(* Logix 5000 project; controller RSL5k_18_Template_noLib Emulate 5570 rev 32.11; software revision 32.02; part 9 of 16 *)
(* tags used below, declared in another part *)
   Inp_CascSP : ALIAS FOR Wrk_PIDE.SPCascade;   // Setpoint in Cascade, Independent PV in Ratio (PVEU)
   Inp_FF : REAL;   // FeedForward term (CVEU)
   Inp_FFPrev : REAL;   // Previous scan FF term (CVEU)
   Inp_CVInitVal : ALIAS FOR Wrk_PIDE.CVInitValue;   // Value to Initialize the CV to when requested (CVRaw)
   Inp_CVPrev : REAL;   // Previous scan CV (CVEU)
   Inp_UseCVInitVal : ALIAS FOR Wrk_PIDE.CVInitReq;   // 1=Initialize CV to Inp_CVInitValue
   Inp_HandFdbk : REAL;   // CV Feedback used in Hand Mode (CVEU)
   Inp_OvrdRatio : REAL;   // Loop Ratio in Override (unitless)
   Inp_OvrdSP : REAL;   // Loop Auto Setpoint (SP) in Override (PVEU)
   Inp_OvrdCV : REAL;   // Loop Manual Output (CV) in Override (CVEU)
   Inp_OvrdSPRoCLimInc : REAL;   // Override Setting for Setpoint Positive Rate of Change Limit (PVEU/sec)
   Inp_OvrdSPRoCLimDec : REAL;   // Override Setting for Setpoint Negative Rate of Change Limit (PVEU/sec)
   Cfg_HasRatio : ALIAS FOR Wrk_PIDE.UseRatio;   // 1=Casc Loop Mode is Ratio, 0=Casc Loop Mode is Cascade
   Cfg_PVTrack : ALIAS FOR Wrk_PIDE.PVTracking;   // 1=SP tracks PV in Manual, 0=no PV tracking
   Cfg_LimitManCV : ALIAS FOR Wrk_PIDE.CVManLimiting;   // 1=CV limits enforced in Manual, 0=No CV Limiting in Manual
   Cfg_SetTrack : BOOL;   // 1=Prog/Oper/Ext Settings track, 0=no Settings tracking
   Cfg_SetTrackOvrdHand : BOOL;   // 1=Prog/Oper/Ext Settings track Override/Hand Inputs (CV, SP, Ratio)
   Cfg_SkipSPRoCLim : BOOL;   // 1=Skip SP RoC Limiting in Intlk, Maint, Ovrd
   Cfg_NormLM : DINT;   // Normal Loop Mode 0=Disable Normal selection, 1=Man, 2=Auto, 3=Casc
   Cfg_PwrupLM : DINT;   // Powerup Loop Mode 0=No change (last), 1=Man (w/ CV), 2=Auto (w/ SP), 3=Casc, 4=Normal
   Cfg_IntlkTripCVAct : DINT;   // Interlock Trip CV Action: 0=none, 1=hold last good, 2=use Cfg_IntlkCV
   Cfg_SPFailCVAct : DINT;   // SP Fail CV Action: 0=none, 1=hold last good, 2=use Cfg_IntlkCV
   Cfg_PVFailCVAct : DINT;   // PV Fail CV Action: 1=hold last good, 2=use Cfg_IntlkCV
   Cfg_CVFailCVAct : DINT;   // CV Fail CV Action: 1=hold last good, 2=use Cfg_IntlkCV
   Cfg_MinSP : ALIAS FOR Wrk_PIDE.SPLLimit;   // Minimum allowed Setpoint (SP) (PVEU)
   Cfg_MaxSP : ALIAS FOR Wrk_PIDE.SPHLimit;   // Maximum allowed Setpoint (SP) (PVEU)
   Cfg_MaxSPRoCInc : REAL;   // Maximum allowed Setpoint Positive Rate of Change Limit (PVEU/sec)
   Cfg_MaxSPRoCDec : REAL;   // Maximum allowed Setpoint Negative Rate of Change Limit (PVEU/sec)
   Cfg_SPRampMaxDev : REAL;   // If deviation exceeds this value, pause SP ramp (0.0=never pause) (PVEU)
   Cfg_PVEUMin : ALIAS FOR Wrk_PIDE.PVEUMin;   // PV Engineering Units Mimimum Value (PVEU)
   Cfg_PVEUMax : ALIAS FOR Wrk_PIDE.PVEUMax;   // PV Engineering Units Maximum Value (PVEU)
   Cfg_CVEUMin : REAL;   // CV Engineering Units Minimum Value (CVEU)
   Cfg_CVEUMax : REAL;   // CV Engineering Units Maximum Value (CVEU)
   Cfg_CVRawMin : ALIAS FOR Wrk_PIDE.CVEUMin;   // CV Output Units Minimum Value (CVRaw, for scaling))
   Cfg_CVRawMax : ALIAS FOR Wrk_PIDE.CVEUMax;   // CV Output Units Maximum Value (CVRaw, for scaling)
   Cfg_ExecT : REAL;   // Execution Time (interval) for PID Algorithm (sec)
   Cfg_MinCV : REAL;   // Minimum allowed Controlled Variable (CV) value (CVEU)
   Cfg_MaxCV : REAL;   // Maximum allowed Controlled Variable (CV) value (CVEU)
   Cfg_CVRoCLim : REAL;   // CV Rate of Change Limit (CVEU/sec)
   Cfg_MaxInactiveCV : REAL;   // When Val_CV is greater than this value, set Sts_Active (for HMI) (CVEU)
   Cfg_IntlkCV : REAL;   // CV Value to use with Interlock / Bad Value CV action (CVEU)
   Cfg_PwrupCV : REAL;   // Loop CV on powerup, used if Cfg_PwrupLM <> 0 (none) (CVEU)
   PSet_Ratio : REAL;   // Program Setting for Ratio (loop CasRat and Ratio enabled) (unitless)
   PSet_SP : REAL;   // Program Setting for Setpoint (loop Auto) (PVEU)
   PSet_SPRoCLimInc : REAL;   // Program Setting for Setpoint Rate of Change Limit Increasing (PVEU/sec)
   PSet_SPRoCLimDec : REAL;   // Program Setting for Setpoint Rate of Change Limit Decreasing (PVEU/sec)
   PSet_CV : REAL;   // Program Setting for Controlled Variable (loop Manual) (CVEU)
   XSet_Ratio : REAL;   // External Setting for Ratio (loop CasRat and Ratio enabled) (unitless)
   XSet_SP : REAL;   // External Setting for Setpoint (loop Auto) (PVEU)
   XSet_SPRoCLimInc : REAL;   // External Setting for Setpoint Rate of Change Limit Increasing (PVEU/sec)
   XSet_SPRoCLimDec : REAL;   // External Setting for Setpoint Rate of Change Limit Decreasing (PVEU/sec)
   XSet_CV : REAL;   // External Setting for Controlled Variable (loop Manual) (CVEU)
   Out_CV : ALIAS FOR Wrk_PIDE.CVEU;   // CV to final control element (CV Raw Units)
   Val_PV : REAL;   // Value of Loop PV (PVEU)
   Val_Ratio : ALIAS FOR Wrk_PIDE.Ratio;   // Value of Loop Ratio (unitless)
   Val_SPSet : REAL;   // Value of selected SP (before clamping and ramping) (PVEU)
   Val_SPRoCInc : REAL;   // Current Value of Setpoint Rate of Change Limit Increasing (PVEU/sec)
   Val_SPRoCDec : REAL;   // Current Value of Setpoint Rate of Change Limit Decreasing (PVEU/sec)
   Val_E : ALIAS FOR Wrk_PIDE.E;   // Loop Error (PV-SP) (PVEU)
   Val_CVSet : REAL;   // Value of selected CV (before clamping and ramping) (CVEU)
   Val_CVOut : REAL;   // Value of CV Output (after ramping and clamping (CVEU)
   Val_ActExecT : ALIAS FOR Wrk_PIDE.DeltaT;   // Actual PID Algorithm Execution Time (Interval) (sec)
   Val_Init : REAL;   // Initialization Value for this loop's Cascade Primary (PVEU)
   Val_PVEUMin : REAL;   // Minimum of PV scaled range (PVEU)
   Val_PVEUMax : REAL;   // Maximum of PV scaled range (PVEU)
   Val_CVEUMin : REAL;   // Minimum of CV scaled range (CVEU)
   Val_CVEUMax : REAL;   // Maximum of CV scaled range (CVEU)
   Sts_InstrFaults1 : DINT;   // PIDE Block Status1 Instruction Fault bits (See PIDE Instruction Help)
   Sts_InstrFaults2 : DINT;   // PIDE Block Status2 Instruction Fault bits (See PIDE Instruction Help)
   Sts_Casc : BOOL;   // 1=Loop Mode is Cascade/Ratio
   Sts_Auto : BOOL;   // 1=Loop Mode is Auto
   Sts_Man : BOOL;   // 1=Loop Mode is Manual
   Sts_NormLM : BOOL;   // 1=Loop is in Normal Loop Mode (see Cfg_NormLM)
   Sts_InitReq : BOOL;   // 1=CV Initialize Request to this loop's Primary
   Sts_RatioClamped : BOOL;   // 1=Selected Ratio (PSet/OSet_Ratio or Inp_OvrdRatio) has been clamped
   Sts_SPBad : ALIAS FOR Wrk_PIDE.SPProgInv;   // 1=SP Value is Bad (quality) or invalid or Casc SP comms fault
   Sts_IntlkSP : BOOL;   // 1=SP Value is being set by shed to Interlock SP
   Sts_SPHeld : BOOL;   // 1=SP Value is being set by shed to hold last good SP
   Sts_SPShed : BOOL;   // 1=SP from Shed, 0=SP from Prog, Oper, Ovrd (A), Casc SP Input (C) or PV Track (M)
   Sts_SPTrackPV : BOOL;   // 1=SP Value is being set by PV Tracking (in Manual Mode)
   Sts_SPClamped : BOOL;   // 1=Selected SP is being clamped (for faceplate animation)
   Sts_SPRamping : BOOL;   // 1=SP is ramping toward Val_SPSet, 0=ramp complete
   Sts_SkipSPRoCLim : BOOL;   // 1=SP rate limiting is being skipped (for faceplate animation)
   Sts_PVBad : BOOL;   // 1=PV Value, comms, quality or EU Limitis Bad
   Sts_CVBad : BOOL;   // 1=CV Value is Bad (quality) or invalid or CV comms fault
   Sts_IntlkCV : BOOL;   // 1=CV Value is being set by shed to Interlock CV
   Sts_CVHeld : BOOL;   // 1=CV Value is being set by shed to hold last good CV
   Sts_CVShed : BOOL;   // 1=CV from Shed, 0=CV from Prog, Oper, Ovrd (Man), or PID (Auto, Casc)
   Sts_CVClamped : BOOL;   // 1=Selected CV is being clamped (for faceplate animation)
   Sts_Active : BOOL;   // 1=CV is greater than Cfg_MaxInactiveCV, show graphic symbol as "active"
   Sts_Err : BOOL;   // 1=Error in Config: see detail Err bits for reason
   Err_Timer : BOOL;   // 1=Error in Config: Status On-Delay or Off-Delay Time Invalid
   Err_RatioLim : ALIAS FOR Wrk_PIDE.RatioLimitsInv;   // 1=Error in Config: Ratio Clamping Limits Invalid
   Err_SPLim : ALIAS FOR Wrk_PIDE.SPLimitsInv;   // 1=Error in Config: Setpoint Clamping Limits Invalid
   Err_CVLim : ALIAS FOR Wrk_PIDE.CVLimitsInv;   // 1=Error in Config: CV Clamping Limits Invalid
   Err_PVEU : ALIAS FOR Wrk_PIDE.PVSpanInv;   // 1=Error in Config: PV EU Max/Min Invalid
   Err_CVEU : BOOL;   // 1=Error in Config: CV EU Max/Min Invalid
   Sts_Hand : ALIAS FOR CmdSrc.Sts_Hand;
   Sts_OoS : ALIAS FOR CmdSrc.Sts_OoS;
   Sts_Maint : ALIAS FOR CmdSrc.Sts_Maint;
   Sts_Ovrd : ALIAS FOR CmdSrc.Sts_Ovrd;
   Sts_Fail : ALIAS FOR Fail.Inp;   // 1=Loop Failure: PV Bad, SP Bad or CV Comm Failure or Bad
   P_PIDE : BOOL;   // Unique Parameter Name for auto - discovery
   CmdSrc : P_CmdSrc;   // Control / Command Source Selection
   Fail : P_Alarm;   // Loop (SP, PV or CV) Failure Alarm
   Wrk_ScanTime : REAL;   // Time since previous scan (sec)
   Wrk_SPStepInc : REAL;   // Amount to add this scan for SP RoC increasing limiting (PVEU)
   Wrk_ScanT : TIMER;   // Scan Timer (milliseconds, always runs)
   Wrk_Casc : BOOL;   // Internal Loop Mode latch: Cascade selected
   Wrk_Auto : BOOL;   // Internal Loop Mode latch: 1=Auto selected
   Wrk_Man : BOOL;   // Internal Loop Mode latch: Manual selected
   Wrk_SPStepDec : REAL;   // Amount to add this scan for SP RoC decreasing limiting (PVEU)
   Wrk_IntlkTripShed : BOOL;   // Shed Latch for Interlock Not OK
   Wrk_PVFailShed : BOOL;   // Shed Latch for PV Failure
   Wrk_SPFailShed : BOOL;   // Shed Latch for SP Failure
   Wrk_CVFailShed : BOOL;   // Shed Latch for CV Failure
   Wrk_AlgoScanT : REAL;   // Time since last calculation of PID Algorithm (sec)
   Wrk_SkippedPID : BOOL;   // PID Algorithm was NOT scanned this time through
   LoLoDevGate : P_Gate;   // Low-Low Deviation Gate/Delay
   LoDevGate : P_Gate;   // Low Deviation Gate/Delay
   HiDevGate : P_Gate;   // High Deviation Gate/Delay
   HiHiDevGate : P_Gate;   // High-High Deviation Gate/Delay
   Wrk_PIDE : PID_ENHANCED;   // Built-in controller PID algorithm
   Wrk_Autotune : PIDE_AUTOTUNE;   // Autotune tag associated with built-in PID algorithm
   Wrk_PIDE_only : P_PIDE_only;   // Backing tag for AOI containing PIDE (with optional autotune)
   HMI_HasAutotune : BOOL;   // 1=P_PIDE_Only AOI has been modified to include Autotune par. on PIDE block
   OSet_CV : REAL;   // Operator Setting for Controlled Variable (loop Manual) (CVEU)
   OSet_SPRoCLimDec : REAL;   // Operator Setting for Setpoint Rate of Change Limit Decreasing (PVEU/sec)
   OSet_SPRoCLimInc : REAL;   // Operator Setting for Setpoint Rate of Change Limit Increasing (PVEU/sec)
   OSet_SP : REAL;   // Operator Setting for Setpoint (loop Auto) (PVEU)
   OSet_Ratio : REAL;   // Operator Setting for Ratio (loop CasRat and Ratio enabled) (unitless)
   Wrk_ExtHas : SINT;   // External owns: .0=LM, .1=CV, .2=SP, .3=Ratio
   Wrk_ProgHas : SINT;   // Program owns: .0=LM, .1=CV, .2=SP, .3=Ratio
   Wrk_OperHas : SINT;   // Operator owns: .0=LM, .1=CV, .2=SP, .3=Ratio
   ORdy_CV : BOOL;   // 1=Ready for OSet_CV (enables data entry field)
   ORdy_SP : BOOL;   // 1=Ready for OSet_SP (enables data entry field)
   Wrk_FirstPIDCalc : BOOL;   // PID Not Skipped ONS store
   ORdy_SPRoCLimInc : BOOL;   // 1=Ready for OSet_SPRoCLimInc (enables data entry field)
   ORdy_SPRoCLimDec : BOOL;   // 1=Ready for OSet_SPRoCLimDec (enables data entry field)
   Wrk_Init : BOOL;   // 1=AOI has been initialized
   Wrk_SPRoCLimDec : REAL;   // Actual SP Rate of Change Limit Decreasing
   Wrk_SPRoCLimInc : REAL;   // Actual SP Rate of Change Limit Increasing
   Wrk_SPRampBusy : BOOL;   // 1=SP Ramp Wizard ramp is in progress
   Wrk_RatioClamped : BOOL;   // Buffer for building Sts_RatioClamped
(* P_PIDE, continued *)

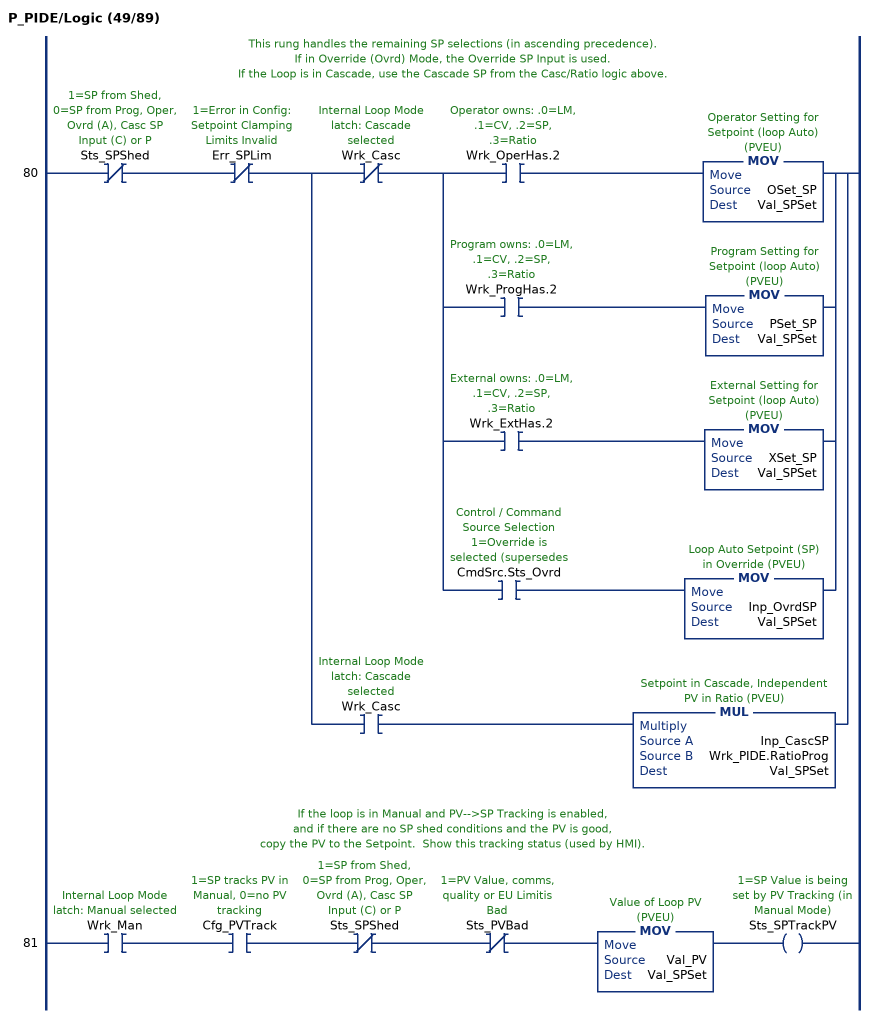
   [picture p175: P_PIDE/Logic rungs 80-81]
   // This rung handles the remaining SP selections (in ascending precedence).
   // If in Override (Ovrd) Mode, the Override SP Input is used.
   // If the Loop is in Cascade, use the Cascade SP from the Casc/Ratio logic above.
   80: XIO(Sts_SPShed)XIO(Err_SPLim)[XIO(Wrk_Casc) [XIC(Wrk_OperHas.2) MOV(OSet_SP,Val_SPSet) ,XIC(Wrk_ProgHas.2) MOV(PSet_SP,Val_SPSet) ,XIC(Wrk_ExtHas.2) MOV(XSet_SP,Val_SPSet) ,XIC(CmdSrc.Sts_Ovrd) MOV(Inp_OvrdSP,Val_SPSet) ] ,XIC(Wrk_Casc) MUL(Inp_CascSP,Wrk_PIDE.RatioProg,Val_SPSet) ];
   // If the loop is in Manual and PV-->SP Tracking is enabled,
   // and if there are no SP shed conditions and the PV is good,
   // copy the PV to the Setpoint.  Show this tracking status (used by HMI).
   81: XIC(Wrk_Man)XIC(Cfg_PVTrack)XIO(Sts_SPShed)XIO(Sts_PVBad)MOV(Val_PV,Val_SPSet)OTE(Sts_SPTrackPV);
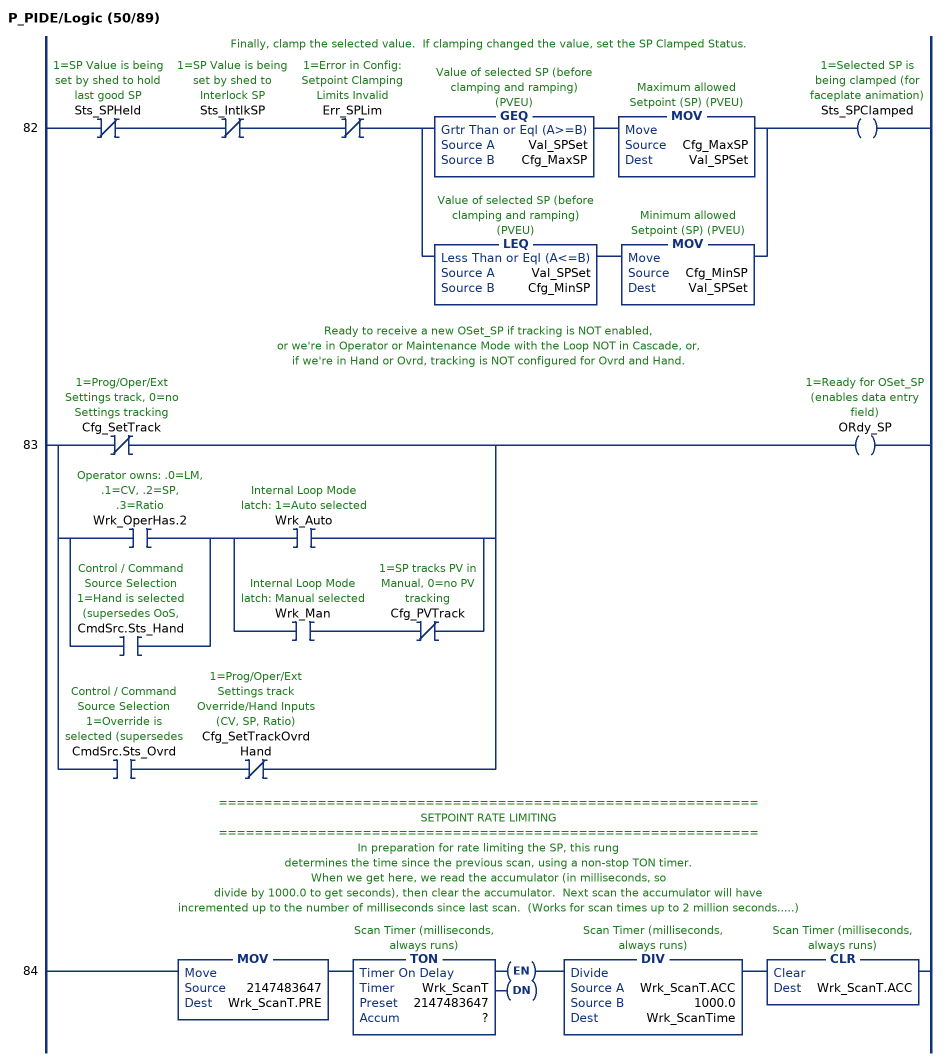
   // Finally, clamp the selected value.  If clamping changed the value, set the SP Clamped Status.
   82: XIO(Sts_SPHeld)XIO(Sts_IntlkSP)XIO(Err_SPLim)[GEQ(Val_SPSet,Cfg_MaxSP) MOV(Cfg_MaxSP,Val_SPSet) ,LEQ(Val_SPSet,Cfg_MinSP) MOV(Cfg_MinSP,Val_SPSet) ]OTE(Sts_SPClamped);
   // Ready to receive a new OSet_SP if tracking is NOT enabled,
   // or we're in Operator or Maintenance Mode with the Loop NOT in Cascade, or,
   // if we're in Hand or Ovrd, tracking is NOT configured for Ovrd and Hand.
   83: [XIO(Cfg_SetTrack) ,[XIC(Wrk_OperHas.2) ,XIC(CmdSrc.Sts_Hand) ] [XIC(Wrk_Auto) ,XIC(Wrk_Man) XIO(Cfg_PVTrack) ] ,XIC(CmdSrc.Sts_Ovrd) XIO(Cfg_SetTrackOvrdHand) ]OTE(ORdy_SP);
   // ============================================================
   // SETPOINT RATE LIMITING
   // ============================================================
   // In preparation for rate limiting the SP, this rung
   // determines the time since the previous scan, using a non-stop TON timer.
   // When we get here, we read the accumulator (in milliseconds, so
   // divide by 1000.0 to get seconds), then clear the accumulator.  Next scan the accumulator will have
   // incremented up to the number of milliseconds since last scan.  (Works for scan times up to 2 million seconds.....)
   84: MOV(2147483647,Wrk_ScanT.PRE)TON(Wrk_ScanT,?,?)DIV(Wrk_ScanT.ACC,1000.0,Wrk_ScanTime)CLR(Wrk_ScanT.ACC);
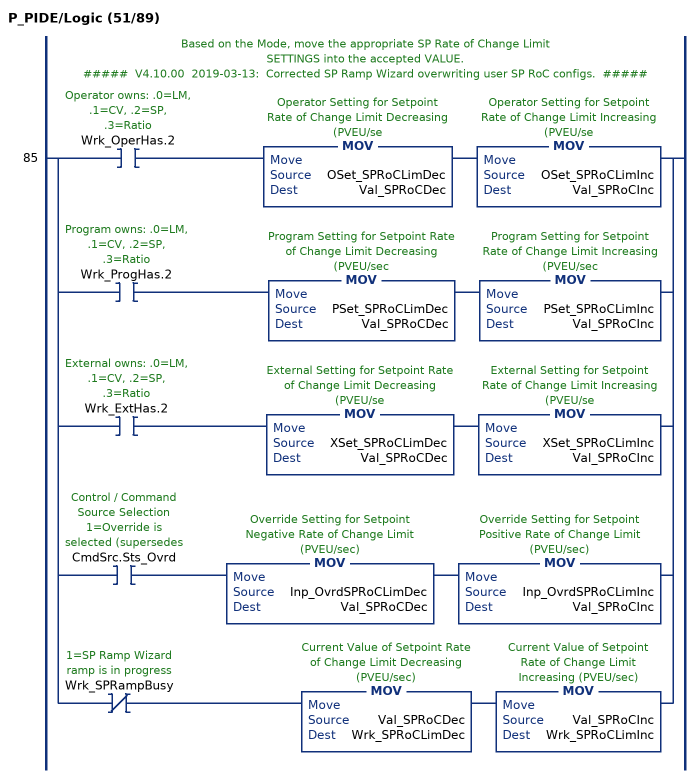
   // Based on the Mode, move the appropriate SP Rate of Change Limit
   // SETTINGS into the accepted VALUE.
   // #####  V4.10.00  2019-03-13:  Corrected SP Ramp Wizard overwriting user SP RoC configs.  #####
   85: [XIC(Wrk_OperHas.2) MOV(OSet_SPRoCLimDec,Val_SPRoCDec) MOV(OSet_SPRoCLimInc,Val_SPRoCInc) ,XIC(Wrk_ProgHas.2) MOV(PSet_SPRoCLimDec,Val_SPRoCDec) MOV(PSet_SPRoCLimInc,Val_SPRoCInc) ,XIC(Wrk_ExtHas.2) MOV(XSet_SPRoCLimDec,Val_SPRoCDec) MOV(XSet_SPRoCLimInc,Val_SPRoCInc) ,XIC(CmdSrc.Sts_Ovrd) MOV(Inp_OvrdSPRoCLimDec,Val_SPRoCDec) MOV(Inp_OvrdSPRoCLimInc,Val_SPRoCInc) ,XIO(Wrk_SPRampBusy) MOV(Val_SPRoCDec,Wrk_SPRoCLimDec) MOV(Val_SPRoCInc,Wrk_SPRoCLimInc) ];
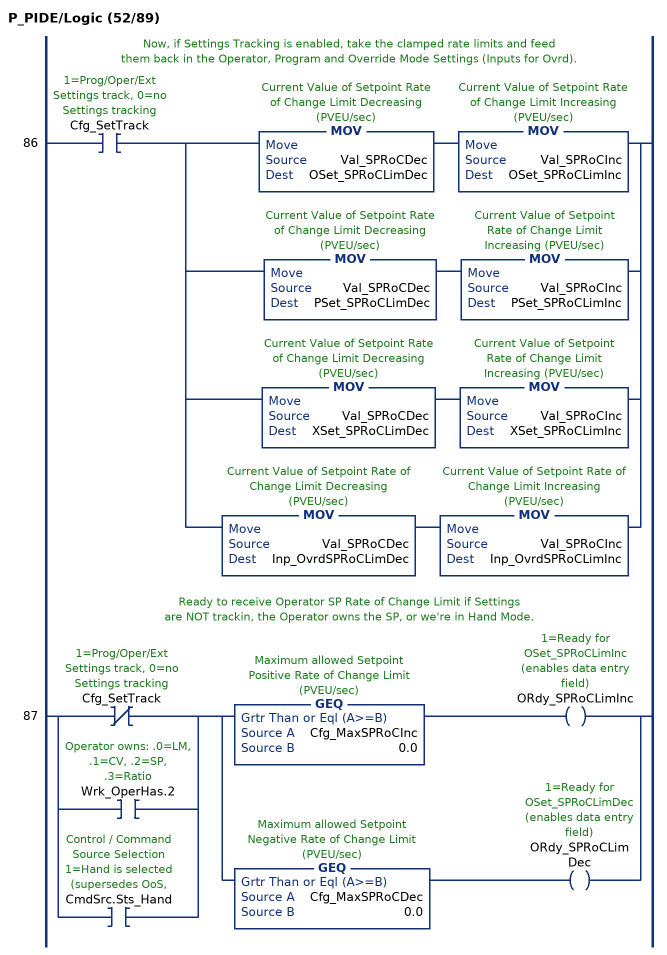
   // Now, if Settings Tracking is enabled, take the clamped rate limits and feed
   // them back in the Operator, Program and Override Mode Settings (Inputs for Ovrd).
   86: XIC(Cfg_SetTrack)[MOV(Val_SPRoCDec,OSet_SPRoCLimDec) MOV(Val_SPRoCInc,OSet_SPRoCLimInc) ,MOV(Val_SPRoCDec,PSet_SPRoCLimDec) MOV(Val_SPRoCInc,PSet_SPRoCLimInc) ,MOV(Val_SPRoCDec,XSet_SPRoCLimDec) MOV(Val_SPRoCInc,XSet_SPRoCLimInc) ,MOV(Val_SPRoCDec,Inp_OvrdSPRoCLimDec) MOV(Val_SPRoCInc,Inp_OvrdSPRoCLimInc) ];
   // Ready to receive Operator SP Rate of Change Limit if Settings
   // are NOT trackin, the Operator owns the SP, or we're in Hand Mode.
   87: [XIO(Cfg_SetTrack) ,XIC(Wrk_OperHas.2) ,XIC(CmdSrc.Sts_Hand) ][GEQ(Cfg_MaxSPRoCInc,0.0) OTE(ORdy_SPRoCLimInc) ,GEQ(Cfg_MaxSPRoCDec,0.0) OTE(ORdy_SPRoCLimDec) ];
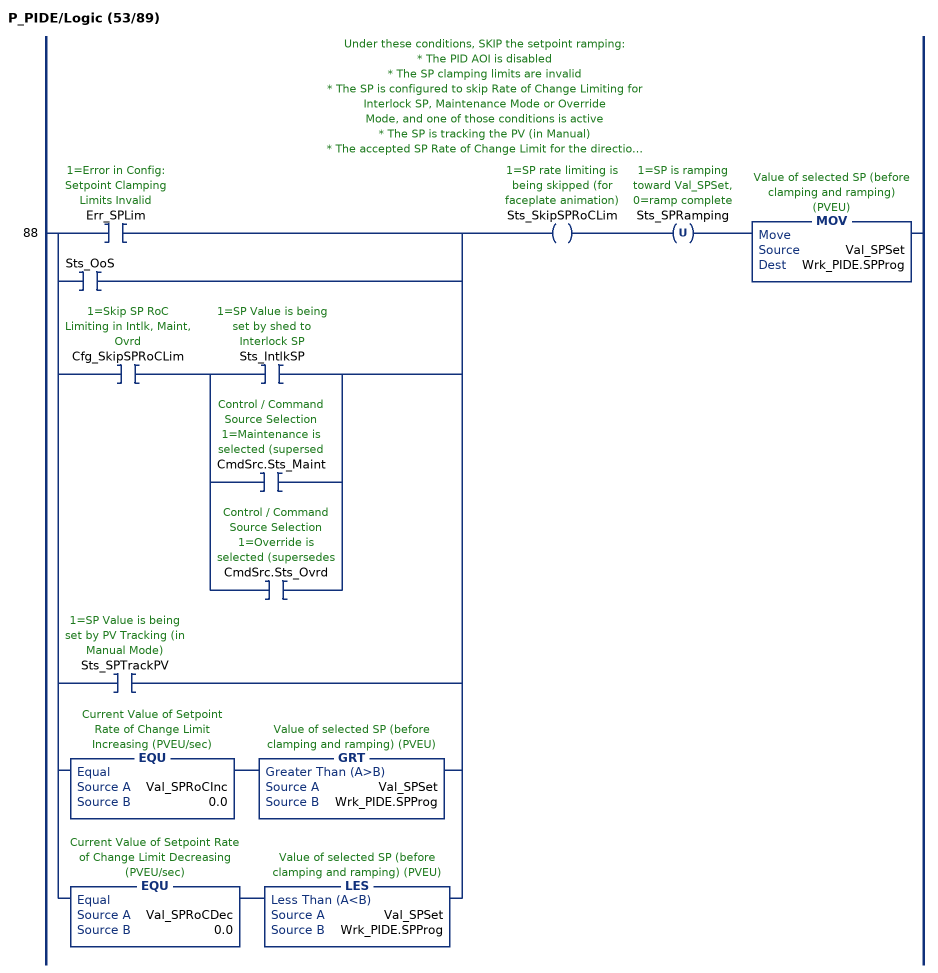
   // Under these conditions, SKIP the setpoint ramping:
   // * The PID AOI is disabled
   // * The SP clamping limits are invalid
   // * The SP is configured to skip Rate of Change Limiting for
   // Interlock SP, Maintenance Mode or Override
   // Mode, and one of those conditions is active
   // * The SP is tracking the PV (in Manual)
   // * The accepted SP Rate of Change Limit for the direction
   // of change (given the error) is ZERO.
   88: [XIC(Err_SPLim) ,XIC(Sts_OoS) ,XIC(Cfg_SkipSPRoCLim) [XIC(Sts_IntlkSP) ,XIC(CmdSrc.Sts_Maint) ,XIC(CmdSrc.Sts_Ovrd) ] ,XIC(Sts_SPTrackPV) ,EQU(Val_SPRoCInc,0.0) GRT(Val_SPSet,Wrk_PIDE.SPProg) ,EQU(Val_SPRoCDec,0.0) LES(Val_SPSet,Wrk_PIDE.SPProg) ]OTE(Sts_SkipSPRoCLim)OTU(Sts_SPRamping)MOV(Val_SPSet,Wrk_PIDE.SPProg);
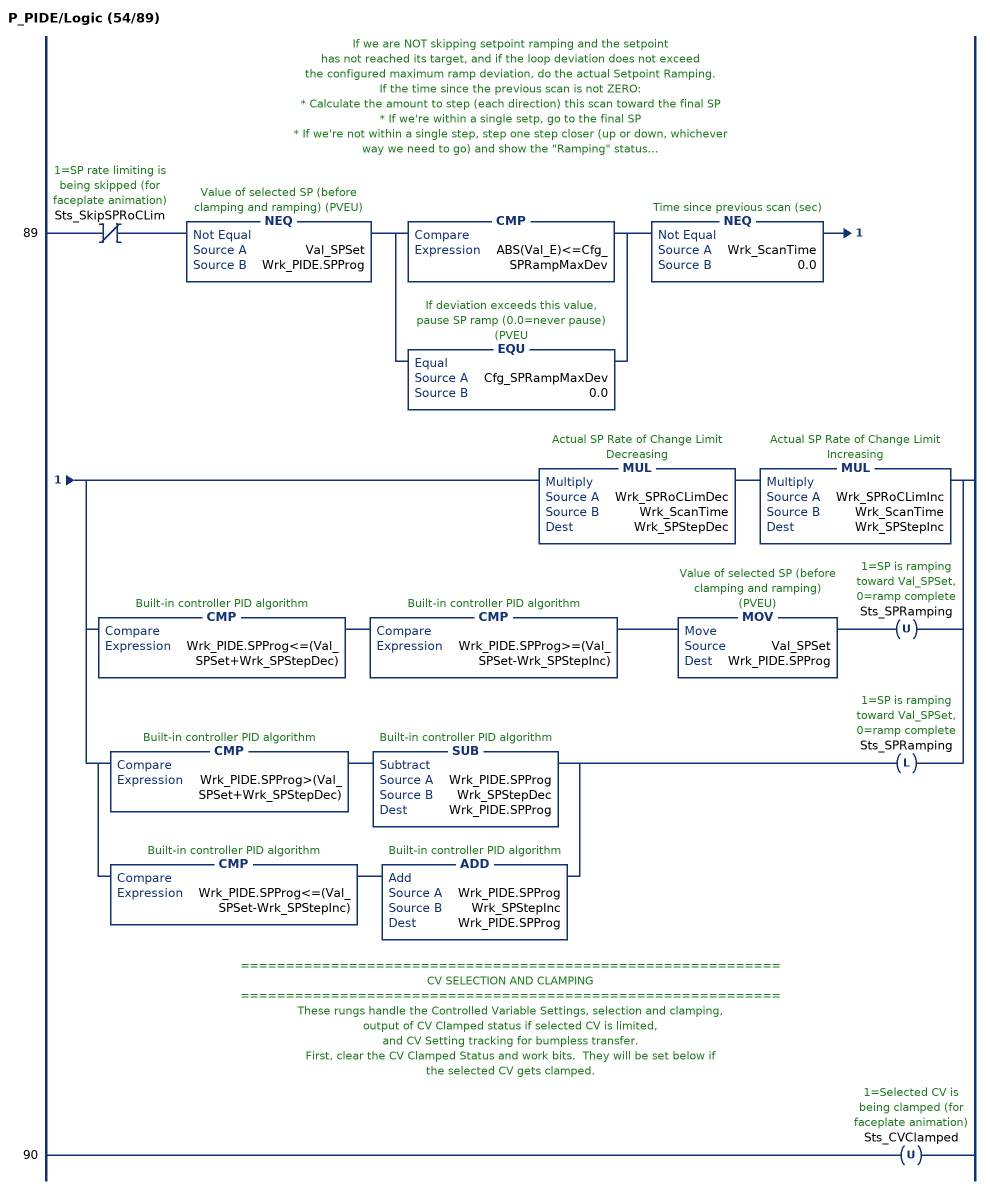
   // If we are NOT skipping setpoint ramping and the setpoint
   // has not reached its target, and if the loop deviation does not exceed
   // the configured maximum ramp deviation, do the actual Setpoint Ramping.
   // If the time since the previous scan is not ZERO:
   // * Calculate the amount to step (each direction) this scan toward the final SP
   // * If we're within a single setp, go to the final SP
   // * If we're not within a single step, step one step closer (up or down, whichever
   // way we need to go) and show the "Ramping" status.
   // #####  V4.10.00  2019-03-13:  Corrected SP Ramp Wizard overwriting user SP RoC configs.  #####
   89: XIO(Sts_SkipSPRoCLim)NEQ(Val_SPSet,Wrk_PIDE.SPProg)[CMP(ABS(Val_E)<=Cfg_SPRampMaxDev) ,EQU(Cfg_SPRampMaxDev,0.0) ]NEQ(Wrk_ScanTime,0.0)[MUL(Wrk_SPRoCLimDec,Wrk_ScanTime,Wrk_SPStepDec) MUL(Wrk_SPRoCLimInc,Wrk_ScanTime,Wrk_SPStepInc) ,CMP(Wrk_PIDE.SPProg<=(Val_SPSet+Wrk_SPStepDec)) CMP(Wrk_PIDE.SPProg>=(Val_SPSet-Wrk_SPStepInc)) MOV(Val_SPSet,Wrk_PIDE.SPProg) OTU(Sts_SPRamping) ,[CMP(Wrk_PIDE.SPProg>(Val_SPSet+Wrk_SPStepDec)) SUB(Wrk_PIDE.SPProg,Wrk_SPStepDec,Wrk_PIDE.SPProg) ,CMP(Wrk_PIDE.SPProg<=(Val_SPSet-Wrk_SPStepInc)) ADD(Wrk_PIDE.SPProg,Wrk_SPStepInc,Wrk_PIDE.SPProg) ] OTL(Sts_SPRamping) ];
   // ============================================================
   // CV SELECTION AND CLAMPING
   // ============================================================
   // These rungs handle the Controlled Variable Settings, selection and clamping,
   // output of CV Clamped status if selected CV is limited,
   // and CV Setting tracking for bumpless transfer.
   // First, clear the CV Clamped Status and work bits.  They will be set below if
   // the selected CV gets clamped.
   90: OTU(Sts_CVClamped);
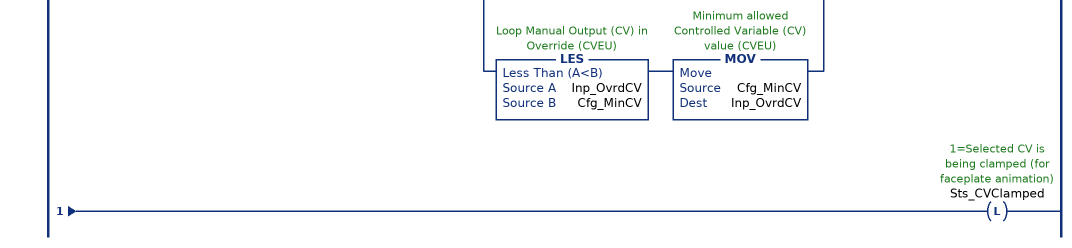
   // This rung handles clamping of the Settings for CV.
   // The value is clamped if necessary here, whether it is used below or not).
   // On the next rung, for the selected Command Source, its CV setting is moved to Val_CVSet.
   // #####  V4.00.01  2018-08-29:  Override Command Source operation.  #####
   // #####  V4.10.01  2019-10-17:  New rung, CVSet selection logic separated from clamping, above.  #####
   91: XIO(Err_CVLim)XIC(Wrk_Man)[[[GRT(PSet_CV,Cfg_CVEUMax) MOV(Cfg_CVEUMax,PSet_CV) ,LES(PSet_CV,Cfg_CVEUMin) MOV(Cfg_CVEUMin,PSet_CV) ] ,XIC(Cfg_LimitManCV) [GRT(PSet_CV,Cfg_MaxCV) MOV(Cfg_MaxCV,PSet_CV) ,LES(PSet_CV,Cfg_MinCV) MOV(Cfg_MinCV,PSet_CV) ] ] XIC(Wrk_ProgHas.1) ,[[GRT(OSet_CV,Cfg_CVEUMax) MOV(Cfg_CVEUMax,OSet_CV) ,LES(OSet_CV,Cfg_CVEUMin) MOV(Cfg_CVEUMin,OSet_CV) ] ,XIC(Cfg_LimitManCV) [GRT(OSet_CV,Cfg_MaxCV) MOV(Cfg_MaxCV,OSet_CV) ,LES(OSet_CV,Cfg_MinCV) MOV(Cfg_MinCV,OSet_CV) ] ] XIC(Wrk_OperHas.1) ,[[GRT(XSet_CV,Cfg_CVEUMax) MOV(Cfg_CVEUMax,XSet_CV) ,LES(XSet_CV,Cfg_CVEUMin) MOV(Cfg_CVEUMin,XSet_CV) ] ,XIC(Cfg_LimitManCV) [GRT(XSet_CV,Cfg_MaxCV) MOV(Cfg_MaxCV,XSet_CV) ,LES(XSet_CV,Cfg_MinCV) MOV(Cfg_MinCV,XSet_CV) ] ] XIC(Wrk_ExtHas.1) ,[[GRT(Inp_OvrdCV,Cfg_CVEUMax) MOV(Cfg_CVEUMax,Inp_OvrdCV) ,LES(Inp_OvrdCV,Cfg_CVEUMin) MOV(Cfg_CVEUMin,Inp_OvrdCV) ] ,XIC(Cfg_LimitManCV) [GRT(Inp_OvrdCV,Cfg_MaxCV) MOV(Cfg_MaxCV,Inp_OvrdCV) ,LES(Inp_OvrdCV,Cfg_MinCV) MOV(Cfg_MinCV,Inp_OvrdCV) ] ] XIC(Sts_Ovrd) ]OTL(Sts_CVClamped);
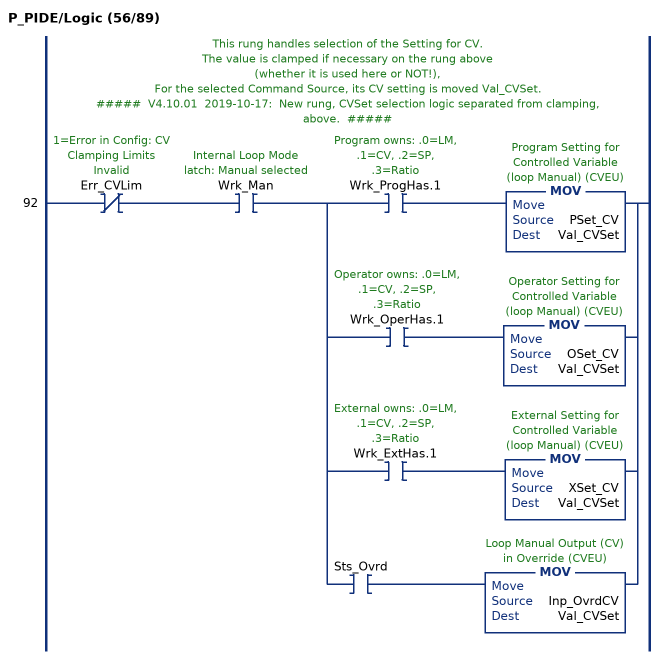
   // This rung handles selection of the Setting for CV.
   // The value is clamped if necessary on the rung above
   // (whether it is used here or NOT!),
   // For the selected Command Source, its CV setting is moved Val_CVSet.
   // #####  V4.10.01  2019-10-17:  New rung, CVSet selection logic separated from clamping, above.  #####
   92: XIO(Err_CVLim)XIC(Wrk_Man)[XIC(Wrk_ProgHas.1) MOV(PSet_CV,Val_CVSet) ,XIC(Wrk_OperHas.1) MOV(OSet_CV,Val_CVSet) ,XIC(Wrk_ExtHas.1) MOV(XSet_CV,Val_CVSet) ,XIC(Sts_Ovrd) MOV(Inp_OvrdCV,Val_CVSet) ];
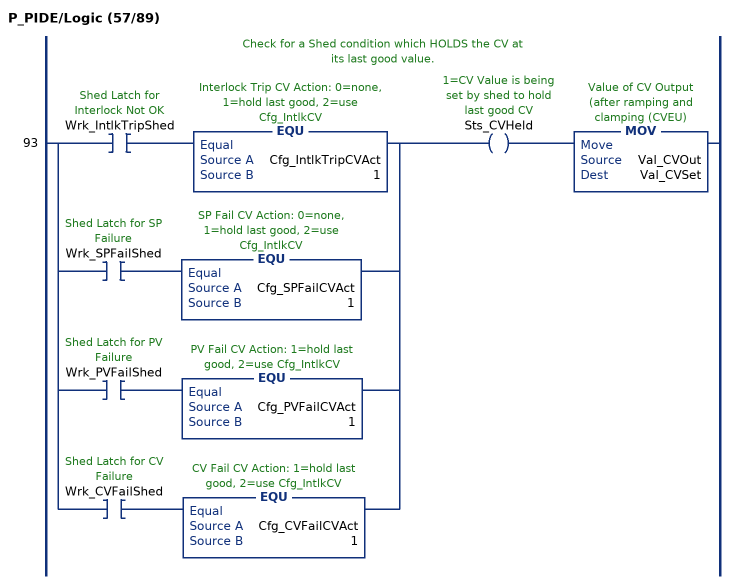
   // Check for a Shed condition which HOLDS the CV at
   // its last good value.
   93: [XIC(Wrk_IntlkTripShed) EQU(Cfg_IntlkTripCVAct,1) ,XIC(Wrk_SPFailShed) EQU(Cfg_SPFailCVAct,1) ,XIC(Wrk_PVFailShed) EQU(Cfg_PVFailCVAct,1) ,XIC(Wrk_CVFailShed) EQU(Cfg_CVFailCVAct,1) ]OTE(Sts_CVHeld)MOV(Val_CVOut,Val_CVSet);
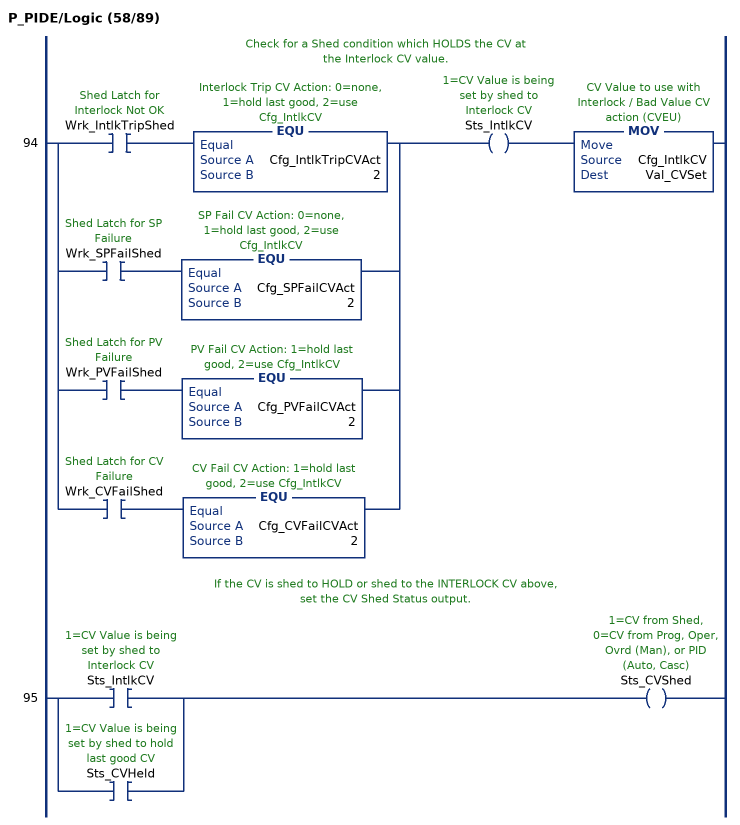
   // Check for a Shed condition which HOLDS the CV at
   // the Interlock CV value.
   94: [XIC(Wrk_IntlkTripShed) EQU(Cfg_IntlkTripCVAct,2) ,XIC(Wrk_SPFailShed) EQU(Cfg_SPFailCVAct,2) ,XIC(Wrk_PVFailShed) EQU(Cfg_PVFailCVAct,2) ,XIC(Wrk_CVFailShed) EQU(Cfg_CVFailCVAct,2) ]OTE(Sts_IntlkCV)MOV(Cfg_IntlkCV,Val_CVSet);
   // If the CV is shed to HOLD or shed to the INTERLOCK CV above,
   // set the CV Shed Status output.
   95: [XIC(Sts_IntlkCV) ,XIC(Sts_CVHeld) ]OTE(Sts_CVShed);
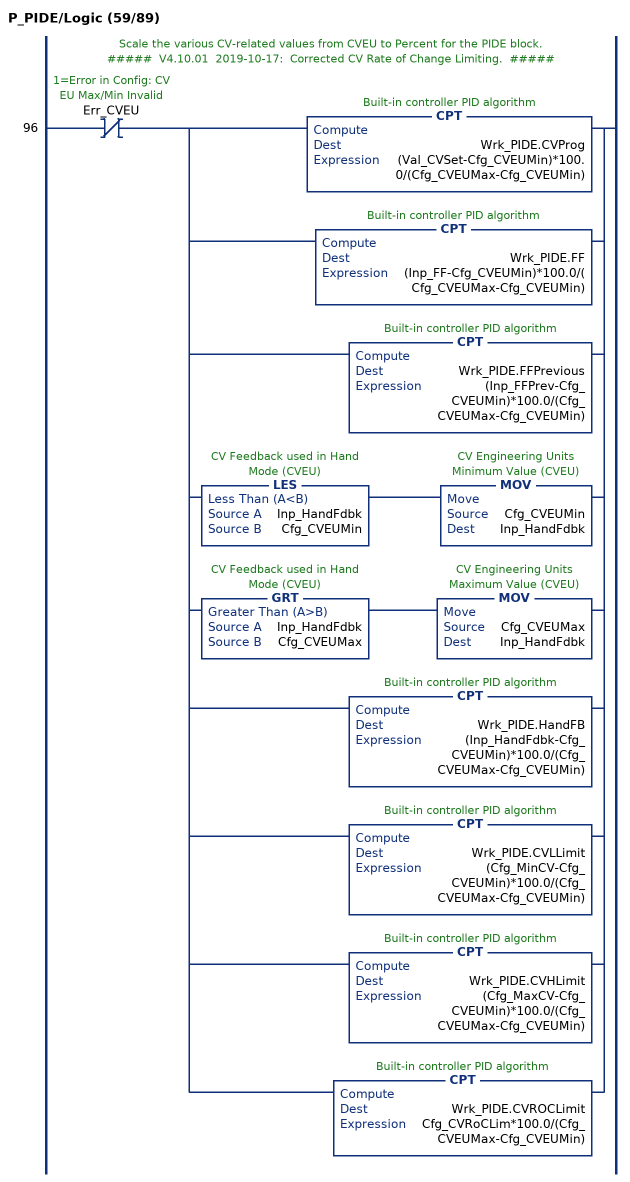
   // Scale the various CV-related values from CVEU to Percent for the PIDE block.
   // #####  V4.10.01  2019-10-17:  Corrected CV Rate of Change Limiting.  #####
   96: XIO(Err_CVEU)[CPT(Wrk_PIDE.CVProg,(Val_CVSet-Cfg_CVEUMin)*100.0/(Cfg_CVEUMax-Cfg_CVEUMin)) ,CPT(Wrk_PIDE.FF,(Inp_FF-Cfg_CVEUMin)*100.0/(Cfg_CVEUMax-Cfg_CVEUMin)) ,CPT(Wrk_PIDE.FFPrevious,(Inp_FFPrev-Cfg_CVEUMin)*100.0/(Cfg_CVEUMax-Cfg_CVEUMin)) ,LES(Inp_HandFdbk,Cfg_CVEUMin) MOV(Cfg_CVEUMin,Inp_HandFdbk) ,GRT(Inp_HandFdbk,Cfg_CVEUMax) MOV(Cfg_CVEUMax,Inp_HandFdbk) ,CPT(Wrk_PIDE.HandFB,(Inp_HandFdbk-Cfg_CVEUMin)*100.0/(Cfg_CVEUMax-Cfg_CVEUMin)) ,CPT(Wrk_PIDE.CVLLimit,(Cfg_MinCV-Cfg_CVEUMin)*100.0/(Cfg_CVEUMax-Cfg_CVEUMin)) ,CPT(Wrk_PIDE.CVHLimit,(Cfg_MaxCV-Cfg_CVEUMin)*100.0/(Cfg_CVEUMax-Cfg_CVEUMin)) ,CPT(Wrk_PIDE.CVROCLimit,Cfg_CVRoCLim*100.0/(Cfg_CVEUMax-Cfg_CVEUMin)) ];
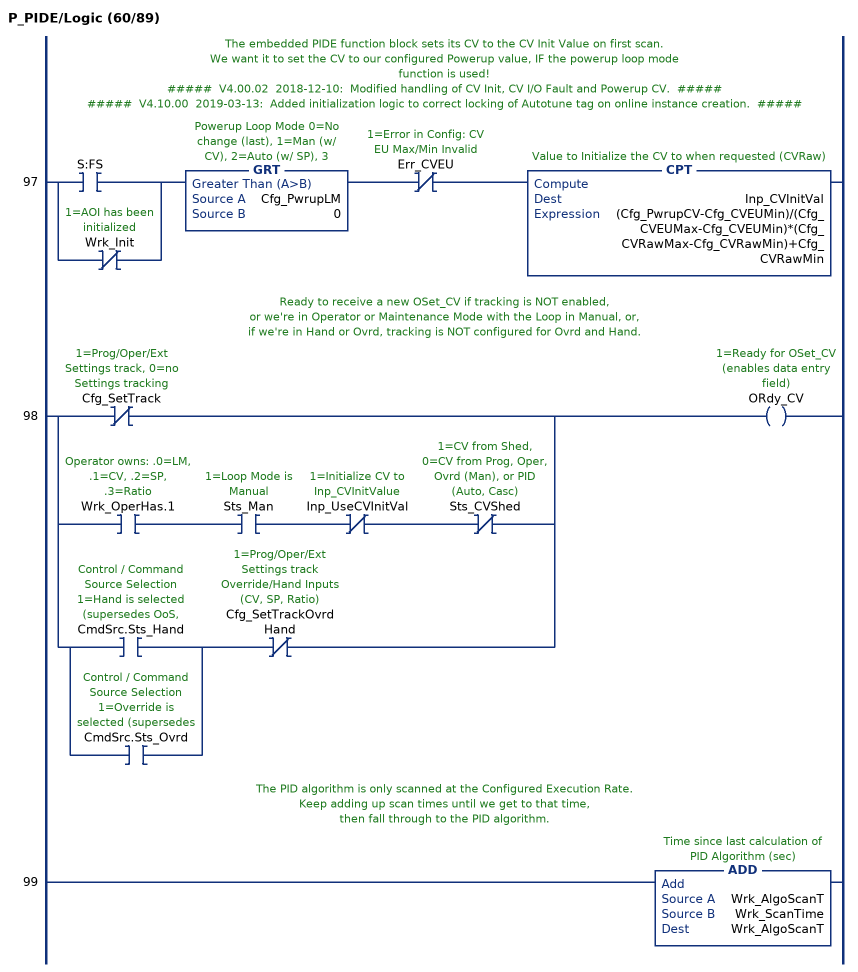
   // The embedded PIDE function block sets its CV to the CV Init Value on first scan.
   // We want it to set the CV to our configured Powerup value, IF the powerup loop mode
   // function is used!
   // #####  V4.00.02  2018-12-10:  Modified handling of CV Init, CV I/O Fault and Powerup CV.  #####
   // #####  V4.10.00  2019-03-13:  Added initialization logic to correct locking of Autotune tag on online instance creation.  #####
   97: [XIC(S:FS) ,XIO(Wrk_Init) ]GRT(Cfg_PwrupLM,0)XIO(Err_CVEU)CPT(Inp_CVInitVal,(Cfg_PwrupCV-Cfg_CVEUMin)/(Cfg_CVEUMax-Cfg_CVEUMin)*(Cfg_CVRawMax-Cfg_CVRawMin)+Cfg_CVRawMin);
   // Ready to receive a new OSet_CV if tracking is NOT enabled,
   // or we're in Operator or Maintenance Mode with the Loop in Manual, or,
   // if we're in Hand or Ovrd, tracking is NOT configured for Ovrd and Hand.
   98: [XIO(Cfg_SetTrack) ,XIC(Wrk_OperHas.1) XIC(Sts_Man) XIO(Inp_UseCVInitVal) XIO(Sts_CVShed) ,[XIC(CmdSrc.Sts_Hand) ,XIC(CmdSrc.Sts_Ovrd) ] XIO(Cfg_SetTrackOvrdHand) ]OTE(ORdy_CV);
   // The PID algorithm is only scanned at the Configured Execution Rate.
   // Keep adding up scan times until we get to that time,
   // then fall through to the PID algorithm.
   99: ADD(Wrk_AlgoScanT,Wrk_ScanTime,Wrk_AlgoScanT);
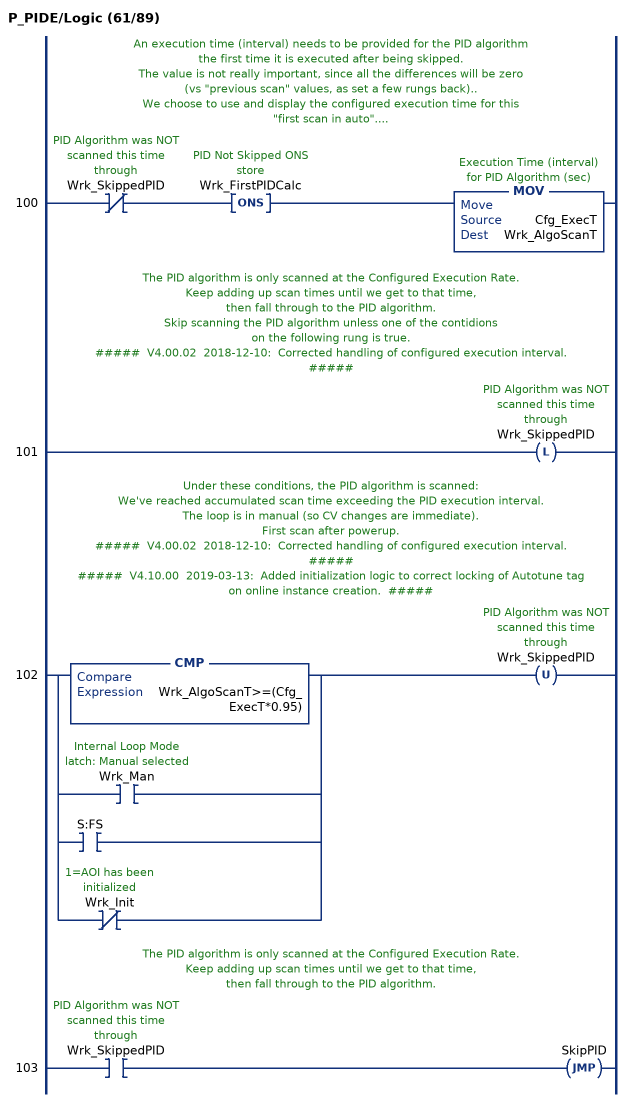
   // An execution time (interval) needs to be provided for the PID algorithm
   // the first time it is executed after being skipped.
   // The value is not really important, since all the differences will be zero
   // (vs "previous scan" values, as set a few rungs back)..
   // We choose to use and display the configured execution time for this
   // "first scan in auto"....
   100: XIO(Wrk_SkippedPID)ONS(Wrk_FirstPIDCalc)MOV(Cfg_ExecT,Wrk_AlgoScanT);
   // The PID algorithm is only scanned at the Configured Execution Rate.
   // Keep adding up scan times until we get to that time,
   // then fall through to the PID algorithm.
   // Skip scanning the PID algorithm unless one of the contidions
   // on the following rung is true.
   // #####  V4.00.02  2018-12-10:  Corrected handling of configured execution interval.  #####
   101: OTL(Wrk_SkippedPID);
   // Under these conditions, the PID algorithm is scanned:
   // We've reached accumulated scan time exceeding the PID execution interval.
   // The loop is in manual (so CV changes are immediate).
   // First scan after powerup.
   // #####  V4.00.02  2018-12-10:  Corrected handling of configured execution interval.  #####
   // #####  V4.10.00  2019-03-13:  Added initialization logic to correct locking of Autotune tag on online instance creation.  #####
   102: [CMP(Wrk_AlgoScanT>=(Cfg_ExecT*0.95)) ,XIC(Wrk_Man) ,XIC(S:FS) ,XIO(Wrk_Init) ]OTU(Wrk_SkippedPID);
   // The PID algorithm is only scanned at the Configured Execution Rate.
   // Keep adding up scan times until we get to that time,
   // then fall through to the PID algorithm.
   103: XIC(Wrk_SkippedPID)JMP(SkipPID);
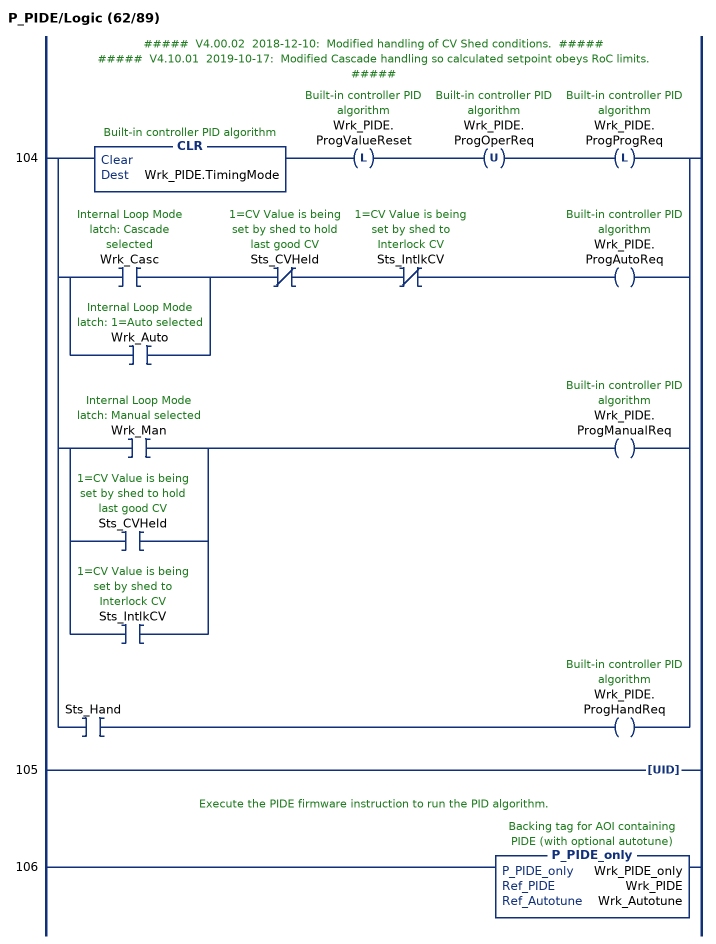
   // #####  V4.00.02  2018-12-10:  Modified handling of CV Shed conditions.  #####
   // #####  V4.10.01  2019-10-17:  Modified Cascade handling so calculated setpoint obeys RoC limits.  #####
   104: [CLR(Wrk_PIDE.TimingMode) OTL(Wrk_PIDE.ProgValueReset) OTU(Wrk_PIDE.ProgOperReq) OTL(Wrk_PIDE.ProgProgReq) ,[XIC(Wrk_Casc) ,XIC(Wrk_Auto) ] XIO(Sts_CVHeld) XIO(Sts_IntlkCV) OTE(Wrk_PIDE.ProgAutoReq) ,[XIC(Wrk_Man) ,XIC(Sts_CVHeld) ,XIC(Sts_IntlkCV) ] OTE(Wrk_PIDE.ProgManualReq) ,XIC(Sts_Hand) OTE(Wrk_PIDE.ProgHandReq) ];
   105: UID();
   // Execute the PIDE firmware instruction to run the PID algorithm.
   106: P_PIDE_only(Wrk_PIDE_only,Wrk_PIDE,Wrk_Autotune);
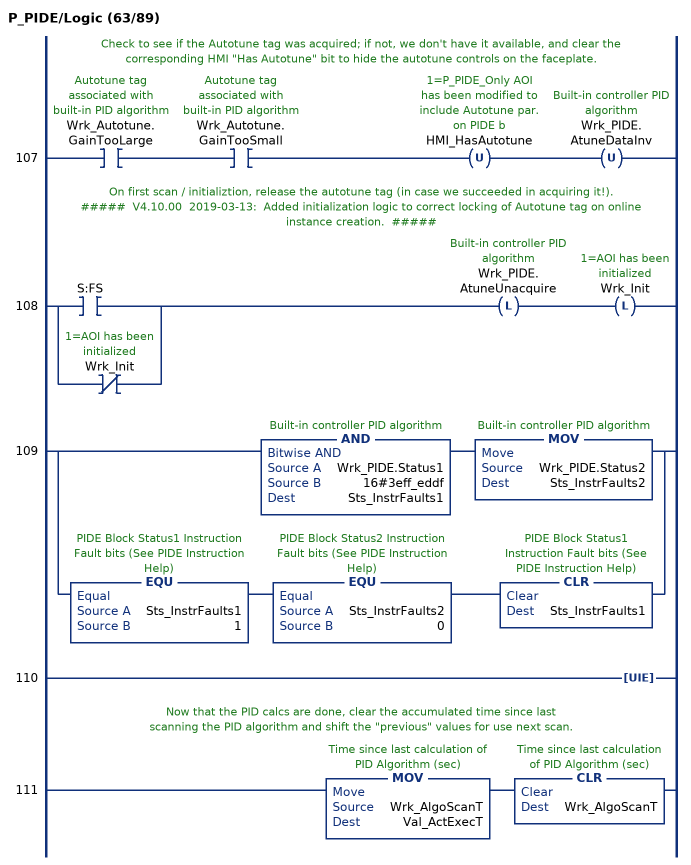
   // Check to see if the Autotune tag was acquired; if not, we don't have it available, and clear the
   // corresponding HMI "Has Autotune" bit to hide the autotune controls on the faceplate.
   107: XIC(Wrk_Autotune.GainTooLarge)XIC(Wrk_Autotune.GainTooSmall)OTU(HMI_HasAutotune)OTU(Wrk_PIDE.AtuneDataInv);
   // On first scan / initializtion, release the autotune tag (in case we succeeded in acquiring it!).
   // #####  V4.10.00  2019-03-13:  Added initialization logic to correct locking of Autotune tag on online instance creation.  #####
   108: [XIC(S:FS) ,XIO(Wrk_Init) ]OTL(Wrk_PIDE.AtuneUnacquire)OTL(Wrk_Init);
   109: [AND(Wrk_PIDE.Status1,16#3eff_eddf,Sts_InstrFaults1) MOV(Wrk_PIDE.Status2,Sts_InstrFaults2) ,EQU(Sts_InstrFaults1,1) EQU(Sts_InstrFaults2,0) CLR(Sts_InstrFaults1) ];
   110: UIE();
   // Now that the PID calcs are done, clear the accumulated time since last
   // scanning the PID algorithm and shift the "previous" values for use next scan.
   111: MOV(Wrk_AlgoScanT,Val_ActExecT)CLR(Wrk_AlgoScanT);
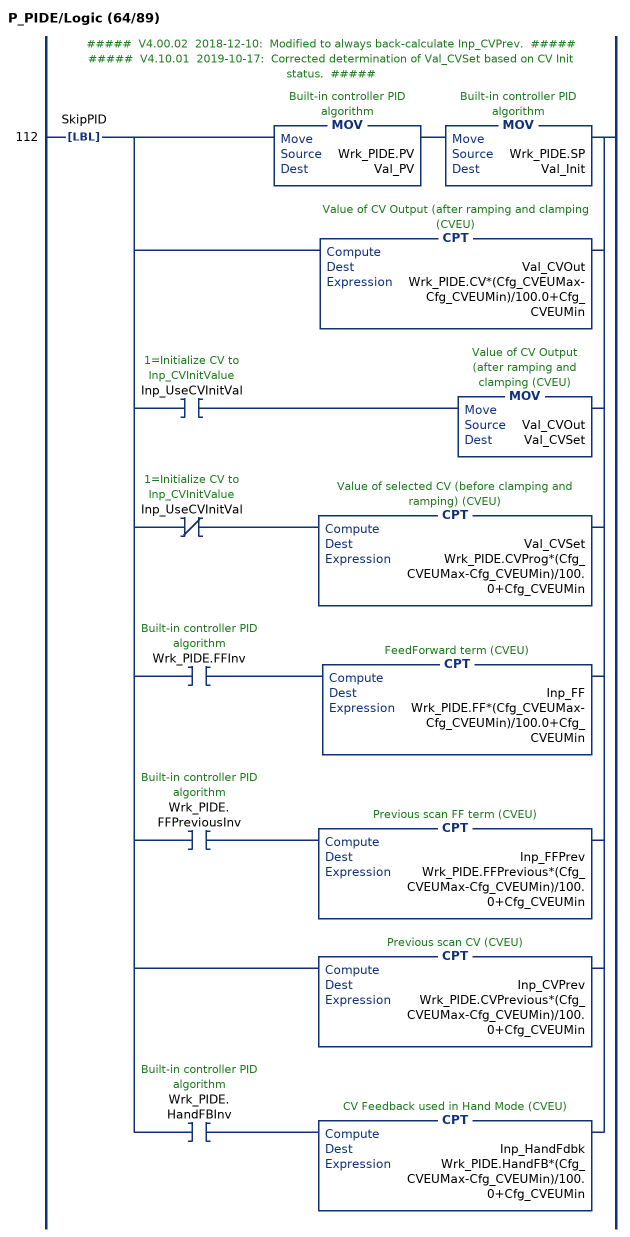
   // #####  V4.00.02  2018-12-10:  Modified to always back-calculate Inp_CVPrev.  #####
   // #####  V4.10.01  2019-10-17:  Corrected determination of Val_CVSet based on CV Init status.  #####
   112: LBL(SkipPID)[MOV(Wrk_PIDE.PV,Val_PV) MOV(Wrk_PIDE.SP,Val_Init) ,CPT(Val_CVOut,Wrk_PIDE.CV*(Cfg_CVEUMax-Cfg_CVEUMin)/100.0+Cfg_CVEUMin) ,XIC(Inp_UseCVInitVal) MOV(Val_CVOut,Val_CVSet) ,XIO(Inp_UseCVInitVal) CPT(Val_CVSet,Wrk_PIDE.CVProg*(Cfg_CVEUMax-Cfg_CVEUMin)/100.0+Cfg_CVEUMin) ,XIC(Wrk_PIDE.FFInv) CPT(Inp_FF,Wrk_PIDE.FF*(Cfg_CVEUMax-Cfg_CVEUMin)/100.0+Cfg_CVEUMin) ,XIC(Wrk_PIDE.FFPreviousInv) CPT(Inp_FFPrev,Wrk_PIDE.FFPrevious*(Cfg_CVEUMax-Cfg_CVEUMin)/100.0+Cfg_CVEUMin) ,CPT(Inp_CVPrev,Wrk_PIDE.CVPrevious*(Cfg_CVEUMax-Cfg_CVEUMin)/100.0+Cfg_CVEUMin) ,XIC(Wrk_PIDE.HandFBInv) CPT(Inp_HandFdbk,Wrk_PIDE.HandFB*(Cfg_CVEUMax-Cfg_CVEUMin)/100.0+Cfg_CVEUMin) ];
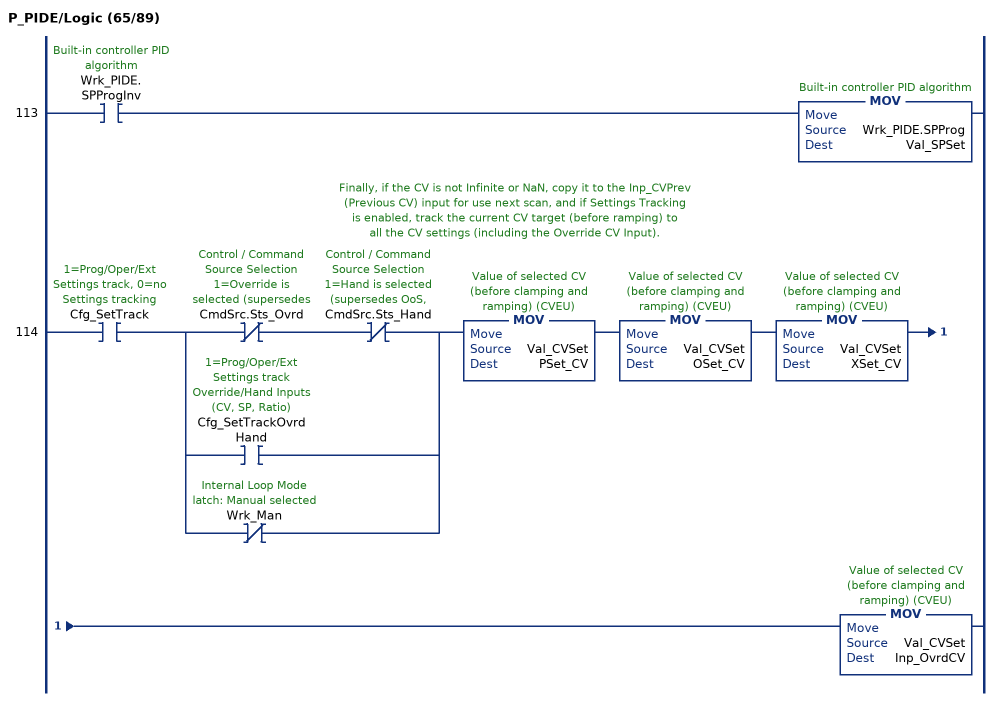
   113: XIC(Wrk_PIDE.SPProgInv)MOV(Wrk_PIDE.SPProg,Val_SPSet);
   // Finally, if the CV is not Infinite or NaN, copy it to the Inp_CVPrev
   // (Previous CV) input for use next scan, and if Settings Tracking
   // is enabled, track the current CV target (before ramping) to
   // all the CV settings (including the Override CV Input).
   114: XIC(Cfg_SetTrack)[[XIO(CmdSrc.Sts_Ovrd) XIO(CmdSrc.Sts_Hand) ,XIC(Cfg_SetTrackOvrdHand) ] ,XIO(Wrk_Man) ]MOV(Val_CVSet,PSet_CV)MOV(Val_CVSet,OSet_CV)MOV(Val_CVSet,XSet_CV)MOV(Val_CVSet,Inp_OvrdCV);
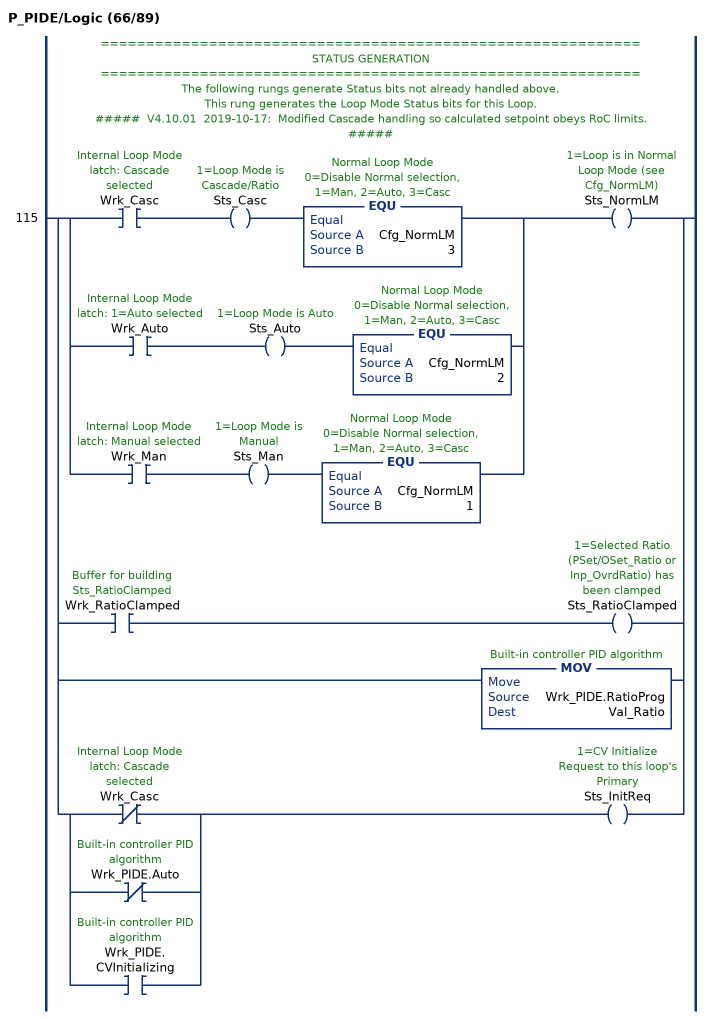
   // ============================================================
   // STATUS GENERATION
   // ============================================================
   // The following rungs generate Status bits not already handled above.
   // This rung generates the Loop Mode Status bits for this Loop.
   // #####  V4.10.01  2019-10-17:  Modified Cascade handling so calculated setpoint obeys RoC limits.  #####
   115: [[XIC(Wrk_Casc) OTE(Sts_Casc) EQU(Cfg_NormLM,3) ,XIC(Wrk_Auto) OTE(Sts_Auto) EQU(Cfg_NormLM,2) ,XIC(Wrk_Man) OTE(Sts_Man) EQU(Cfg_NormLM,1) ] OTE(Sts_NormLM) ,XIC(Wrk_RatioClamped) OTE(Sts_RatioClamped) ,MOV(Wrk_PIDE.RatioProg,Val_Ratio) ,[XIO(Wrk_Casc) ,XIO(Wrk_PIDE.Auto) ,XIC(Wrk_PIDE.CVInitializing) ] OTE(Sts_InitReq) ];
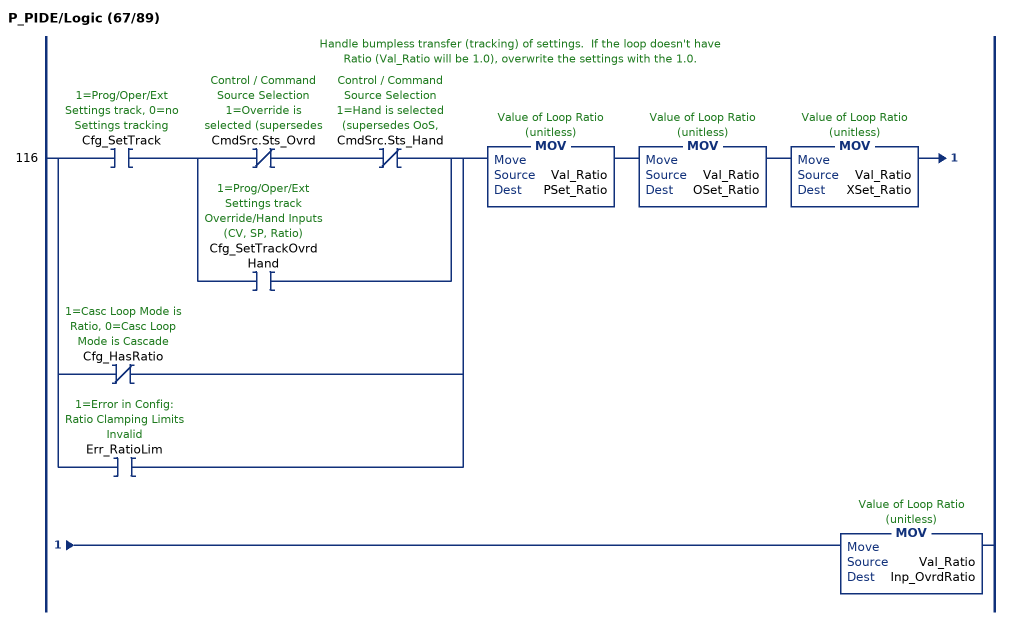
   // Handle bumpless transfer (tracking) of settings.  If the loop doesn't have
   // Ratio (Val_Ratio will be 1.0), overwrite the settings with the 1.0.
   116: [XIC(Cfg_SetTrack) [XIO(CmdSrc.Sts_Ovrd) XIO(CmdSrc.Sts_Hand) ,XIC(Cfg_SetTrackOvrdHand) ] ,XIO(Cfg_HasRatio) ,XIC(Err_RatioLim) ]MOV(Val_Ratio,PSet_Ratio)MOV(Val_Ratio,OSet_Ratio)MOV(Val_Ratio,XSet_Ratio)MOV(Val_Ratio,Inp_OvrdRatio);
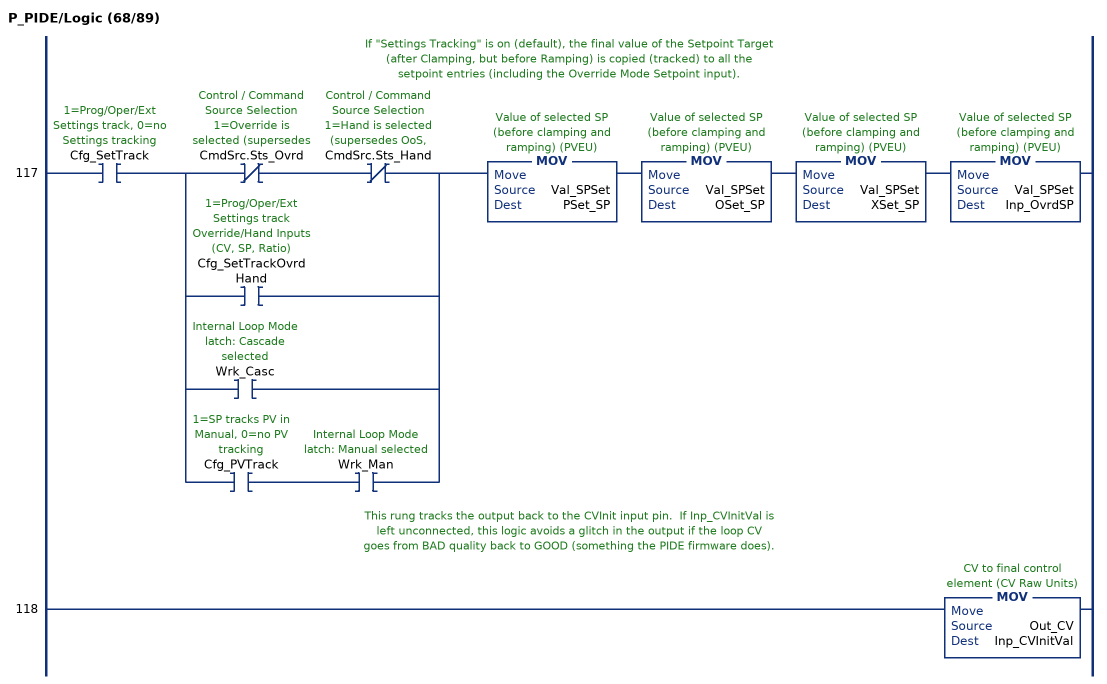
   // If "Settings Tracking" is on (default), the final value of the Setpoint Target
   // (after Clamping, but before Ramping) is copied (tracked) to all the
   // setpoint entries (including the Override Mode Setpoint input).
   117: XIC(Cfg_SetTrack)[[XIO(CmdSrc.Sts_Ovrd) XIO(CmdSrc.Sts_Hand) ,XIC(Cfg_SetTrackOvrdHand) ] ,XIC(Wrk_Casc) ,XIC(Cfg_PVTrack) XIC(Wrk_Man) ]MOV(Val_SPSet,PSet_SP)MOV(Val_SPSet,OSet_SP)MOV(Val_SPSet,XSet_SP)MOV(Val_SPSet,Inp_OvrdSP);
   // This rung tracks the output back to the CVInit input pin.  If Inp_CVInitVal is
   // left unconnected, this logic avoids a glitch in the output if the loop CV
   // goes from BAD quality back to GOOD (something the PIDE firmware does).
   118: MOV(Out_CV,Inp_CVInitVal);
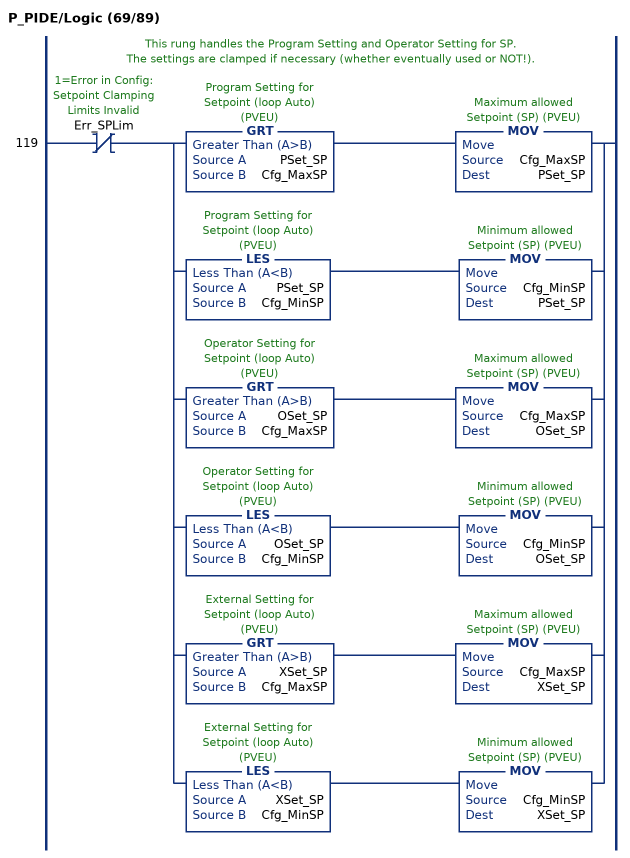
   // This rung handles the Program Setting and Operator Setting for SP.
   // The settings are clamped if necessary (whether eventually used or NOT!).
   119: XIO(Err_SPLim)[GRT(PSet_SP,Cfg_MaxSP) MOV(Cfg_MaxSP,PSet_SP) ,LES(PSet_SP,Cfg_MinSP) MOV(Cfg_MinSP,PSet_SP) ,GRT(OSet_SP,Cfg_MaxSP) MOV(Cfg_MaxSP,OSet_SP) ,LES(OSet_SP,Cfg_MinSP) MOV(Cfg_MinSP,OSet_SP) ,GRT(XSet_SP,Cfg_MaxSP) MOV(Cfg_MaxSP,XSet_SP) ,LES(XSet_SP,Cfg_MinSP) MOV(Cfg_MinSP,XSet_SP) ];
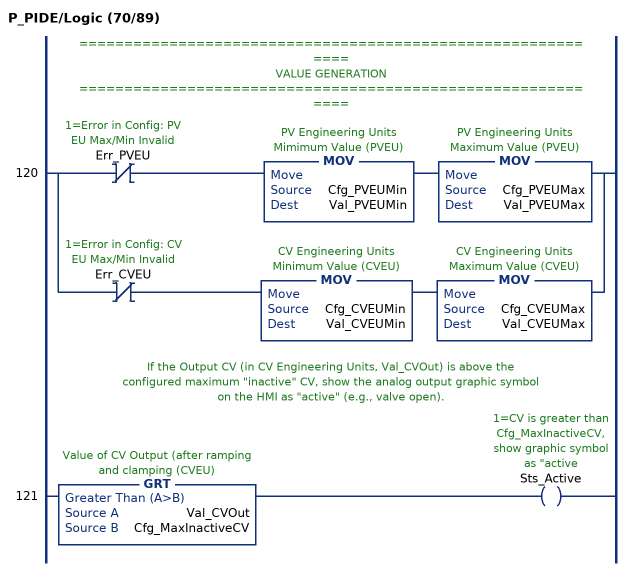
   // ============================================================
   // VALUE GENERATION
   // ============================================================
   120: [XIO(Err_PVEU) MOV(Cfg_PVEUMin,Val_PVEUMin) MOV(Cfg_PVEUMax,Val_PVEUMax) ,XIO(Err_CVEU) MOV(Cfg_CVEUMin,Val_CVEUMin) MOV(Cfg_CVEUMax,Val_CVEUMax) ];
   // If the Output CV (in CV Engineering Units, Val_CVOut) is above the
   // configured maximum "inactive" CV, show the analog output graphic symbol
   // on the HMI as "active" (e.g., valve open).
   121: GRT(Val_CVOut,Cfg_MaxInactiveCV)OTE(Sts_Active);
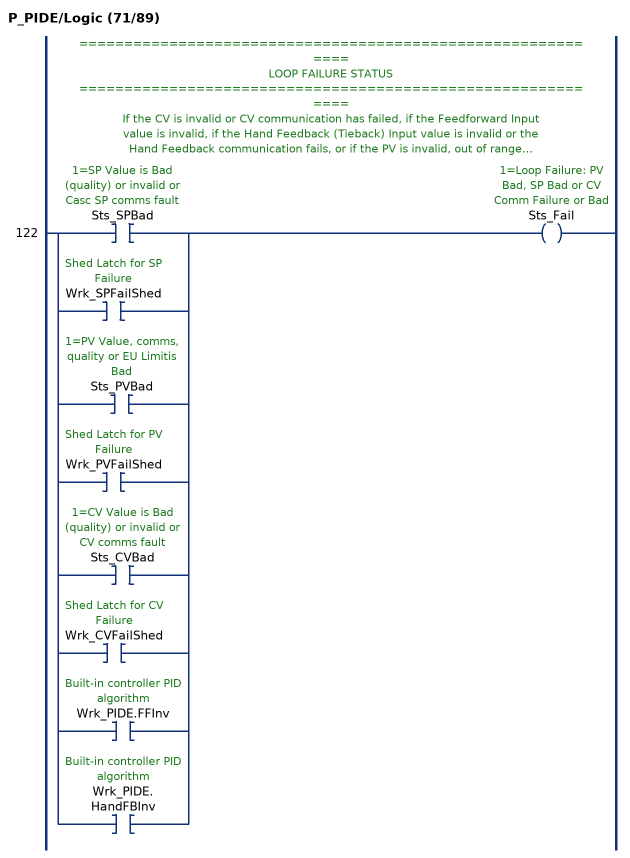
   // ============================================================
   // LOOP FAILURE STATUS
   // ============================================================
   // If the CV is invalid or CV communication has failed, if the Feedforward Input
   // value is invalid, if the Hand Feedback (Tieback) Input value is invalid or the
   // Hand Feedback communication fails, or if the PV is invalid, out of range,
   // bad quality or not being communicated, or if the SP is invalid (or, for
   // cascade, not being communicated),
   // then there is a Loop Failure.  Raise a FAIL STATUS.
   // #####  V4.00.02  2018-12-10:  Modified CV I/O Fault handling, other failure handing.  #####
   122: [XIC(Sts_SPBad) ,XIC(Wrk_SPFailShed) ,XIC(Sts_PVBad) ,XIC(Wrk_PVFailShed) ,XIC(Sts_CVBad) ,XIC(Wrk_CVFailShed) ,XIC(Wrk_PIDE.FFInv) ,XIC(Wrk_PIDE.HandFBInv) ]OTE(Sts_Fail);
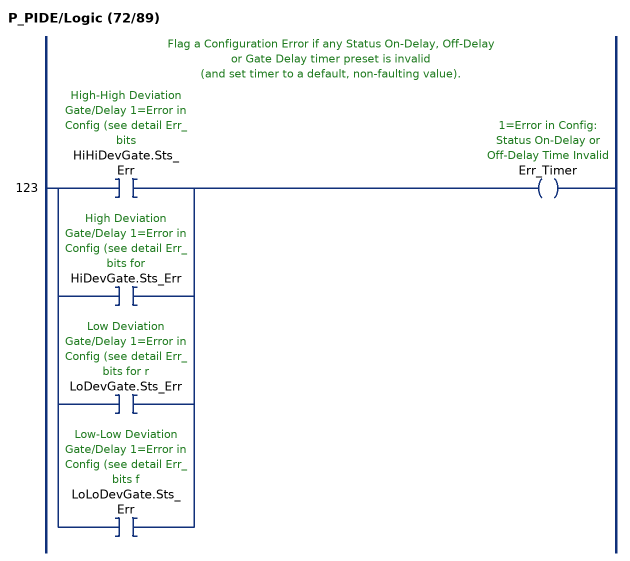
   // Flag a Configuration Error if any Status On-Delay, Off-Delay
   // or Gate Delay timer preset is invalid
   // (and set timer to a default, non-faulting value).
   123: [XIC(HiHiDevGate.Sts_Err) ,XIC(HiDevGate.Sts_Err) ,XIC(LoDevGate.Sts_Err) ,XIC(LoLoDevGate.Sts_Err) ]OTE(Err_Timer);
